// TIA Portal V17 export
// export: Created 2025-07-01T14:26:15.5873158Z, ExportSetting WithDefaults, DisplayName Totally Integrated Automation Portal, DisplayVersion V17 Update 8, DisplayName TIA Portal Openness, DisplayVersion V17 Update 8, DisplayName TIA Portal Version Control Interface, DisplayVersion V17, DisplayName SINAMICS Startdrive Advanced, DisplayVersion V17 SP2, DisplayName SINAMICS Startdrive G110M, G120, G120C, G120D, G120P, G115D, DisplayVersion V17 SP2, DisplayName SINAMICS Startdrive G130, G150, S120, S150, SINAMICS MV, S210, DisplayVersion V17 SP2, DisplayName STEP 7 Professional, DisplayVersion V17 Update 8, DisplayName SINUMERIK ONE STEP 7 Toolbox, DisplayVersion V17 Update 12, DisplayName SINUMERIK ONE PLC Basic Program Plus, DisplayVersion V17 Update 12, DisplayName SINUMERIK 840D sl STEP 7 Toolbox, DisplayVersion V17 Update 12, DisplayName STEP 7 Safety, DisplayVersion V17 Update 6, DisplayName WinCC Advanced, DisplayVersion V17 Update 8
DATA_BLOCK "DB7300_INTERLOCK_GENERAL"   // DB7300
{ S7_Optimized_Access := 'FALSE'; DB_Accessible_From_OPC_UA := 'FALSE' }
AUTHOR : ETXETAR
VERSION : 1.0
// stored: AutoNumber false, DBAccessibleFromOPCUA false, DBAccessibleFromWebserver true, IsOnlyStoredInLoadMemory false, IsWriteProtectedInAS false
   VAR RETAIN
      GENERAL_MACHINE : Struct
         FROM_CELL_TO_MACHINE_GENERAL : Struct
            MEAS_STA_START_CYCLE : Bool;   // CELL MEASURING STATION START CYCLE
            MEAS_STA_CALIB_CYCLE : Bool;   // CELL MEASURING STATION CALIBRATION CYCLE
            MEAS_STA_HOME_REQ : Bool;   // CELL MEASURING STATION HOME REQUEST
            MEAS_STA_FAULT : Bool;   // CELL MEASURING STATION FAULT
            MEAS_STA_RESET : Bool;   // CELL MEASURING STATION RESET
            MEAS_STA_ROBOT_OUT_OF_COLLISION : Bool;
            MEAS_STA_PART_LOADED : Bool;   // CELL MEASURING STATION PART LOADED
            MEAS_STA_PART_UNLOADED : Bool;   // CELL MEASURING STATION PART UNLOADED
            MEAS_STA_SEQ_RUNNING : Bool;   // CELL MEASURING STATION SEQUENCE RUNNING
            CELL_COOLING_DEGRADED_MODE : Bool;   // CELL COOLING DEGRADED MODE
            CELL_STARVED : Bool;   // CELL STARVED
            CELL_BLOCKED : Bool;   // CELL BLOCKED
            CELL_LOADING_ACTIVE : Bool;   // CELL LOADING ACTIVE
            CELL_CALIBRATION_CYCLE_REQUIRED : Bool;   // CELL CALIBRATION CYCLE REQUIRED
         END_STRUCT;
         FROM_ROBOT_TO_UNIT_1 : Struct
            HEARTBEAT : Bool;   // ROBOT HEARTBEAT
            EMERG_STOP_OK : Bool;   // ROBOT EMERGENCY STOP OK
            ROBOT_FAULT : Bool;   // ROBOT FAULT
            SAFETY_DOOR_CLSD_LOCKD : Bool;   // ROBOT SAFETY DOOR CLOSED AND LOCKED
            CELL_EMPTY : Bool;   // ROBOT CELL EMPTY
            IN_SEMIAUTO_MODE : Bool;   // ROBOT SEMIAUTO MODE SELECTED
            IN_MANUAL_MODE : Bool;   // ROBOT MANUAL MODE SELECTED
            IN_AUTO_MODE : Bool;   // ROBOT AUTO MODE SELECTED
            IN_AUTO_CYCLE_RUN : Bool;   // ROBOT CYCLE RUNNING IN AUTOMATIC MODE
            RUN_OUT_REQUEST : Bool;   // ROBOT MACHINE RUN OUT REQUEST
            RUN_OUT_COMPLETED : Bool;   // ROBOT RUN OUT COMPLETED
            SAFETY_DOOR_OPEN_REQ : Bool;   // ROBOT ANY CELL SAFETY DOOR OPEN REQUEST
            OK_TO_OPEN_SAFETY_GATES : Bool;   // ROBOT OK TO OPEN SAFETY GATES
            READY_TO_SERVICE : Bool;   // ROBOT READY TO SERVICE MACHINE
            OUT_OF_COLLISION_MACHINE : Bool;   // ROBOT OUT OF COLLISION MACHINE
            OUT_OF_COLLISION_FIXTURE : Bool;   // ROBOT OUT OF COLLISION FIXTURE
            PART_ENABLED : Bool;   // ROBOT PART ENABLED
            PART_FACE_R_TO_DELIVER : Bool;   // ROBOT PART FACE R TO DELIVER IMMEDIATELY
            PART_FACE_N_TO_DELIVER : Bool;   // ROBOT PART FACE N TO DELIVER IMMEDIATELY
            OUT_OF_PARTS_FACE_R_TO_DELIVER : Bool;   // ROBOT OUT OF PARTS FACE R IN CELL TO DELIVER
            OUT_OF_PARTS_FACE_N_TO_DELIVER : Bool;   // ROBOT OUT OF PARTS FACE N IN CELL TO DELIVER
            PART_LOADED : Bool;   // ROBOT PART LOADED
            PART_UNLOADED : Bool;   // ROBOT PART UNLOADED
            FIX_SKIP_REQ : Bool;   // ROBOT FIXTURE SKIP REQUEST
            PART_TYPE_CHANGE_REQ : Bool;   // ROBOT PART TYPE CHANGE REQUEST
            PART_TYPE : Byte;   // ROBOT PART TYPE
         END_STRUCT;
         FROM_ROBOT_TO_UNIT_2 : Struct
            HEARTBEAT : Bool;   // ROBOT HEARTBEAT
            EMERG_STOP_OK : Bool;   // ROBOT EMERGENCY STOP OK
            ROBOT_FAULT : Bool;   // ROBOT FAULT
            SAFETY_DOOR_CLSD_LOCKD : Bool;   // ROBOT SAFETY DOOR CLOSED AND LOCKED
            CELL_EMPTY : Bool;   // ROBOT CELL EMPTY
            IN_SEMIAUTO_MODE : Bool;   // ROBOT SEMIAUTO MODE SELECTED
            IN_MANUAL_MODE : Bool;   // ROBOT MANUAL MODE SELECTED
            IN_AUTO_MODE : Bool;   // ROBOT AUTO MODE SELECTED
            IN_AUTO_CYCLE_RUN : Bool;   // ROBOT CYCLE RUNNING IN AUTOMATIC MODE
            RUN_OUT_REQUEST : Bool;   // ROBOT MACHINE RUN OUT REQUEST
            RUN_OUT_COMPLETED : Bool;   // ROBOT RUN OUT COMPLETED
            SAFETY_DOOR_OPEN_REQ : Bool;   // ROBOT ANY CELL SAFETY DOOR OPEN REQUEST
            OK_TO_OPEN_SAFETY_GATES : Bool;   // ROBOT OK TO OPEN SAFETY GATES
            READY_TO_SERVICE : Bool;   // ROBOT READY TO SERVICE MACHINE
            OUT_OF_COLLISION_MACHINE : Bool;   // ROBOT OUT OF COLLISION MACHINE
            OUT_OF_COLLISION_FIXTURE : Bool;   // ROBOT OUT OF COLLISION FIXTURE
            PART_ENABLED : Bool;   // ROBOT PART ENABLED
            PART_FACE_R_TO_DELIVER : Bool;   // ROBOT PART FACE R TO DELIVER IMMEDIATELY
            PART_FACE_N_TO_DELIVER : Bool;   // ROBOT PART FACE N TO DELIVER IMMEDIATELY
            OUT_OF_PARTS_FACE_R_TO_DELIVER : Bool;   // ROBOT OUT OF PARTS FACE R IN CELL TO DELIVER
            OUT_OF_PARTS_FACE_N_TO_DELIVER : Bool;   // ROBOT OUT OF PARTS FACE N IN CELL TO DELIVER
            PART_LOADED : Bool;   // ROBOT PART LOADED
            PART_UNLOADED : Bool;   // ROBOT PART UNLOADED
            FIX_SKIP_REQ : Bool;   // ROBOT FIXTURE SKIP REQUEST
            PART_TYPE_CHANGE_REQ : Bool;   // ROBOT PART TYPE CHANGE REQUEST
            PART_TYPE : Byte;   // ROBOT PART TYPE
         END_STRUCT;
      END_STRUCT;
      POWDER_PLC : Struct
         GENERAL : Struct
            LIFE_BIT : Bool;   // LIFE BIT
            SELECTED_ARGON_GAS : Bool;   // SELECTED ARGON GAS
            SELECTED_NITROGEN_GAS : Bool;   // SELECTED NITROGEN GAS
            SELECTED_IMPERIAL_SYSTEM : Bool;   // SELECTED IMPERIAL SYSTEM
            SELECTED_METRIC_SYSTEM : Bool;   // SELECTED METRIC SYSTEM
            POWDER_PLC_AUTO_MODE : Bool;   // POWDER PLC IN AUTO MODE
            POWDER_PLC_MAN_MODE : Bool;   // POWDER PLC IN MANUAL MODE
         END_STRUCT;
         FROM_POWDER_TO_UNIT_1 : Struct
            POWDER_UNIT_1_READY_TO_RUN : Bool;   // POWDER UNIT 1 READY TO RUN
            POWDER_UNIT_1_STOPPED : Bool;   // POWDER UNIT 1 STOPPED
            SWITCHED_ON_POWDER_UNIT_1 : Bool;   // SWITCHED ON POWDER UNIT 1
            SWITCHED_OFF_POWDER_UNIT_1 : Bool;   // SWITCHED OFF POWDER UNIT 1
            SWITCHED_ON_TEMPERATURE_JACKET_UNIT_1 : Bool;   // SWITCHED ON TEMPERATURE JACKET UNIT 1
            SWITCHED_OFF_TEMPERATURE_JACKET_UNIT_1 : Bool;   // SWITCHED OFF TEMPERATURE JACKET UNIT 1
            U1_PF_1_LINE_1_LOW_POWDER : Bool;   // UNIT 1 POWDER FEEDER 1 LINE 1 LOW POWDER LEVEL
            U1_PF_1_LINE_2_LOW_POWDER : Bool;   // UNIT 1 POWDER FEEDER 1 LINE 2 LOW POWDER LEVEL
            POWDER_UNIT_1_ALARM : Bool;   // POWDER UNIT 1 ALARM
            UNIT_1_POWDER_FEEDER_1_CARRIER_GAS_ACTUAL_LINE_1 : Real;   // UNIT 1 POWDER FEEDER 1 CARRIER GAS ACTUAL LINE 1
            UNIT_1_POWDER_FEEDER_1_DISK_SPEED_ACTUAL_LINE_1 : Real;   // UNIT 1 POWDER FEEDER 1 DISK SPEED ACTUAL LINE 1
            UNIT_1_POWDER_FEEDER_1_STIRRER_SPEED_ACTUAL_LINE_1 : Real;   // UNIT 1 POWDER FEEDER 1 STIRRER SPEED ACTUAL LINE 1
            UNIT_1_POWDER_FEEDER_1_HOPPER_TEMPERATURE_ACTUAL_LINE_1 : Real;   // UNIT 1 POWDER FEEDER 1 HOPPER TEMPERATURE ACTUAL LINE 1
            UNIT_1_POWDER_FEEDER_1_CARRIER_GAS_ACTUAL_LINE_2 : Real;   // UNIT 1 POWDER FEEDER 1 CARRIER GAS ACTUAL LINE 2
            UNIT_1_POWDER_FEEDER_1_DISK_SPEED_ACTUAL_LINE_2 : Real;   // UNIT 1 POWDER FEEDER 1 DISK SPEED ACTUAL LINE 2
            UNIT_1_POWDER_FEEDER_1_STIRRER_SPEED_ACTUAL_LINE_2 : Real;   // UNIT 1 POWDER FEEDER 1 STIRRER SPEED ACTUAL LINE 2
            UNIT_1_POWDER_FEEDER_1_HOPPER_TEMPERATURE_ACTUAL_LINE_2 : Real;   // UNIT 1 POWDER FEEDER 1 HOPPER TEMPERATURE ACTUAL LINE 2
         END_STRUCT;
         FROM_POWDER_TO_UNIT_2 : Struct
            POWDER_UNIT_2_READY_TO_RUN : Bool;   // POWDER UNIT 2 READY TO RUN
            POWDER_UNIT_2_STOPPED : Bool;   // POWDER UNIT 2 STOPPED
            SWITCHED_ON_POWDER_UNIT_2 : Bool;   // SWITCHED ON POWDER UNIT 2
            SWITCHED_OFF_POWDER_UNIT_2 : Bool;   // SWITCHED OFF POWDER UNIT 2
            SWITCHED__ON_TEMPERATURE_JACKET_UNIT_2 : Bool;   // SWITCHED ON TEMPERATURE JACKET UNIT 2
            SWITCHED_OFF_TEMPERATURE_JACKET_UNIT_2 : Bool;   // SWITCHED OFF TEMPERATURE JACKET UNIT 2
            U2_PF_1_LINE_1_LOW_POWDER : Bool;   // UNIT 2 POWDER FEEDER 1 LINE 1 LOW POWDER LEVEL
            U2_PF_1_LINE_2_LOW_POWDER : Bool;   // UNIT 2 POWDER FEEDER 1 LINE 2 LOW POWDER LEVEL
            U2_PF_2_LINE_2_LOW_POWDER : Bool;   // UNIT 2 POWDER FEEDER 2 LINE 2 LOW POWDER LEVEL
            POWDER_UNIT_2_ALARM : Bool;   // POWDER UNIT 2 ALARM
            UNIT_2_POWDER_FEEDER_1_CARRIER_GAS_ACTUAL_LINE_1 : Real;   // UNIT 2 POWDER FEEDER 1 CARRIER GAS ACTUAL LINE 1
            UNIT_2_POWDER_FEEDER_1_CARRIER_GAS_ACTUAL_LINE_2 : Real;   // UNIT 2 POWDER FEEDER 1 CARRIER GAS ACTUAL LINE 2
            UNIT_2_POWDER_FEEDER_1_DISK_SPEED_ACTUAL_LINE_1 : Real;   // UNIT 2 POWDER FEEDER 1 DISK SPEED ACTUAL LINE 1
            UNIT_2_POWDER_FEEDER_1_DISK_SPEED_ACTUAL_LINE_2 : Real;   // UNIT 2 POWDER FEEDER 1 DISK SPEED ACTUAL LINE 2
            UNIT_2_POWDER_FEEDER_1_STIRRER_SPEED_ACTUAL_LINE_1 : Real;   // UNIT 2 POWDER FEEDER 1 STIRRER SPEED ACTUAL LINE 1
            UNIT_2_POWDER_FEEDER_1_STIRRER_SPEED_ACTUAL_LINE_2 : Real;   // UNIT 2 POWDER FEEDER 1 STIRRER SPEED ACTUAL LINE 2
            UNIT_2_POWDER_FEEDER_1_HOPPER_TEMPERATURE_ACTUAL_LINE_1 : Real;   // UNIT 2 POWDER FEEDER 1 HOPPER TEMPERATURE ACTUAL LINE 1
            UNIT_2_POWDER_FEEDER_1_HOPPER_TEMPERATURE_ACTUAL_LINE_2 : Real;   // UNIT 2 POWDER FEEDER 1 HOPPER TEMPERATURE ACTUAL LINE 2
            UNIT_2_POWDER_FEEDER_2_CARRIER_GAS_ACTUAL_LINE_1 : Real;   // UNIT 2 POWDER FEEDER 2 CARRIER GAS ACTUAL LINE 1
            UNIT_2_POWDER_FEEDER_2_CARRIER_GAS_ACTUAL_LINE_2 : Real;   // UNIT 2 POWDER FEEDER 2 CARRIER GAS ACTUAL LINE 2
            UNIT_2_POWDER_FEEDER_2_DISK_SPEED_ACTUAL_LINE_1 : Real;   // UNIT 2 POWDER FEEDER 2 DISK SPEED ACTUAL LINE 1
            UNIT_2_POWDER_FEEDER_2_STIRRER_SPEED_ACTUAL_LINE_1 : Real;   // UNIT 2 POWDER FEEDER 2 STIRRER SPEED ACTUAL LINE 1
            UNIT_2_POWDER_FEEDER_2_DISK_SPEED_ACTUAL_LINE_2 : Real;   // UNIT 2 POWDER FEEDER 2 DISK SPEED ACTUAL LINE 2
            UNIT_2_POWDER_FEEDER_2_STIRRER_SPEED_ACTUAL_LINE_2 : Real;   // UNIT 2 POWDER FEEDER 2 STIRRER SPEED ACTUAL LINE 2
            UNIT_2_POWDER_FEEDER_2_HOPPER_TEMPERATURE_ACTUAL_LINE_1 : Real;   // UNIT 2 POWDER FEEDER 2 HOPPER TEMPERATURE ACTUAL LINE 1
            UNIT_2_POWDER_FEEDER_2_HOPPER_TEMPERATURE_ACTUAL_LINE_2 : Real;   // UNIT 2 POWDER FEEDER 2 HOPPER TEMPERATURE ACTUAL LINE 2
         END_STRUCT;
      END_STRUCT;
      LOAD_UNLOAD : Struct
         UNIT_1 : "LOAD_UNLOAD_ETXETAR_ROBOT_CELL";
         UNIT_2 : "LOAD_UNLOAD_ETXETAR_ROBOT_CELL";
         UNIT_3 : "LOAD_UNLOAD_ETXETAR_ROBOT_CELL";
      END_STRUCT;
      AUX_SIGNALS_INTERFACE : Struct
         GENERAL : Struct
            "MEASURING STATION FAULT" : Bool;   // CELL MEASURING STATION FAULT
            "DEGRADED MODE FAULT" : Bool;   // CELL COOLING DEGRADED MODE FAULT
            TIMER_MEASURING_IN_PRCS : TOF_TIME;   // TIMER MEASURING IN PROCESS
            TIMER_MEASURING_DONE : TOF_TIME;   // TIMER MEASURING DONE
         END_STRUCT;
         UNIT_1 : Struct
            LIFE_BIT_FAULT : Bool;   // HEARTBEAT COMMUNICATION ALARM
            EMERGENCY_STOP_ACTIVE : Bool;   // EMERGENCY STOP ACTIVE ALARM
            ROBOT_FAULT_INSIDE_OF_MACHINE : Bool;   // ROBOT FAULT ALARM INSIDE OF MACHINE
            ROBOT_FAULT_OUTSIDE_OF_MACHINE : Bool;   // ROBOT FAULT ALARM OUTSIDE OF MACHINE
            FACE_R_LOAD_REQ_AUX : Bool;   // FACE R LOAD REQUEST AUX
            FACE_N_LOAD_REQ_AUX : Bool;   // FACE N LOAD REQUEST AUX
            "LIFE SING COUNTER" : CTU_INT;
         END_STRUCT;
         UNIT_2 : Struct
            LIFE_BIT_FAULT : Bool;   // HEARTBEAT COMMUNICATION ALARM
            EMERGENCY_STOP_ACTIVE : Bool;   // EMERGENCY STOP ACTIVE ALARM
            ROBOT_FAULT_INSIDE_OF_MACHINE : Bool;   // ROBOT FAULT ALARM INSIDE OF MACHINE
            ROBOT_FAULT_OUTSIDE_OF_MACHINE : Bool;   // ROBOT FAULT ALARM OUTSIDE OF MACHINE
            FACE_R_LOAD_REQ_AUX : Bool;   // FACE R LOAD REQUEST AUX
            FACE_N_LOAD_REQ_AUX : Bool;   // FACE N LOAD REQUEST AUX
            "LIFE SING COUNTER" : CTU_INT;
         END_STRUCT;
         POWDER_PLC : Struct
            LIFE_BIT_FAULT : Bool;   // HEARTBEAT COMMUNICATION ALARM
            "LIFE SING COUNTER" : CTU_INT;
         END_STRUCT;
         AUX_0 : Bool;   // AUXILIARY 0
         AUX_1 : Bool;   // AUXILIARY 1
         AUX_2 : Bool;   // AUXILIARY 2
         AUX_3 : Bool;   // AUXILIARY 3
         AUX_4 : Bool;   // AUXILIARY 4
         AUX_5 : Bool;   // AUXILIARY 5
         AUX_6 : Bool;   // AUXILIARY 6
         AUX_7 : Bool;   // AUXILIARY 7
         AUX_8 : Bool;   // AUXILIARY 8
         AUX_9 : Bool;   // AUXILIARY 9
         AUX_10 : Bool;   // AUXILIARY 10
         AUX_11 : Bool;   // AUXILIARY 11
         AUX_12 : Bool;   // AUXILIARY 12
         AUX_13 : Bool;   // AUXILIARY 13
         AUX_14 : Bool;   // AUXILIARY 14
         AUX_15 : Bool;   // AUXILIARY 15
         TIMER_IS_SEOC_ROBOT_FAULT_UNIT_1 : TON_TIME;   // TIMER IS SEOC ROBOT FAULT UNIT 1
         TIMER_IS_SEOC_ROBOT_FAULT_UNIT_2 : TON_TIME;   // TIMER IS SEOC ROBOT FAULT UNIT 2
         TIMER_SEOC_ROBOT_FAULT_UNIT_1 : TON_TIME;   // TIMER SEOC ROBOT FAULT UNIT 1
         TIMER_SEOC_ROBOT_FAULT_UNIT_2 : TON_TIME;   // TIMER SEOC ROBOT FAULT UNIT 2
      END_STRUCT;
      PART_A : Struct
         UNIT_1 : "PART_STATUS_CLADDING";
         UNIT_2 : "PART_STATUS_CLADDING";
         UNIT_3 : "PART_STATUS_CLADDING";
      END_STRUCT;
   END_VAR
BEGIN
   AUX_SIGNALS_INTERFACE.GENERAL.TIMER_MEASURING_IN_PRCS.PT := T#3s;
   AUX_SIGNALS_INTERFACE.GENERAL.TIMER_MEASURING_DONE.PT := T#3s;
   AUX_SIGNALS_INTERFACE.TIMER_IS_SEOC_ROBOT_FAULT_UNIT_1.PT := T#2M;
   AUX_SIGNALS_INTERFACE.TIMER_IS_SEOC_ROBOT_FAULT_UNIT_2.PT := T#2M;
   AUX_SIGNALS_INTERFACE.TIMER_SEOC_ROBOT_FAULT_UNIT_1.PT := T#2M;
   AUX_SIGNALS_INTERFACE.TIMER_SEOC_ROBOT_FAULT_UNIT_2.PT := T#2M;
END_DATA_BLOCK
